//---------------------------------------------------------------------------------------------------------------
//
//  HAUD 2025.12.29
//
//  - fb_LinkedListCtrl
//  -----------------------------
//  - cyclic wrapper composing fb_LinkedList
//  - used to send tickets over the mapping interfaces
//  . Ctrl / State for you to use
//---------------------------------------------------------------------------------------------------------------
FUNCTION_BLOCK fb_Process_LinkedListCtrl
VAR
  _eCheck             : E_LIST_CHECK;
  _eInit              : E_PROGRESS;

  _eCmd,
  _eCmdOld            : E_LIST_CTRL;
  _eState             : E_LIST_STATE;
  _eResult            : e_progress;

  _ItfList            : I_Process_LinkedList;

  _stCtrl             : REFERENCE TO ST_LIST_CTRL;
  _stState            : REFERENCE TO ST_LIST_STATE;

  _stNodeDataInput    : REFERENCE TO ST_LIST_NODE_DATA;   // datafield for you to write(add) your data
  _stNodeDataOutput   : REFERENCE TO ST_LIST_NODE_DATA;   // datafield for you to read (get) your data

  _stNodeDataProcess  : ST_LIST_NODE_DATA;                // local copy of ProcessData

  _stMsg              : ST_Message;
  _eDevice            : e_Device    := e_device.ProcessListCtrl;     // message device identifier
  _MessageLevel       : E_MessageType;

END_VAR

IF NOT Check() 
THEN
  _eInit                          := E_PROGRESS.PROGRESS_INVALID;
  RETURN; 
END_IF


_eCmd                           := _stCtrl.Cmd;
// check for command change
// get state for cmd
IF (_eCmd <> _eCmdOld)
THEN
  _eState                       := Cmd(_eCmd);
  _eCmdOld                      := _eCmd;

  IF (_MessageLevel > E_MessageType.eMessageError)
  THEN
    _stMsg.eType                := E_MessageType.eMessageInfo;
    _stMsg.eSubdevice           := e_Subdevice.Process_LinkedList_Com;
    _stMsg.iErrorNumber         := 0;
    _stMsg.sText                := concat(TO_STRING(_eCmd), ': ');
    _stMsg.sText                := concat(_stMsg.sText,  TO_STRING(_eState));
    f_MessageSet(_stMsg);
  END_IF
END_IF

CASE _eResult
OF
  E_PROGRESS.PROGRESS_INVALID:
    _stState.State              := TO_UINT(_eResult);

  E_PROGRESS.PROGRESS_ERROR:
    _stState.State              := _eState + E_PROGRESS.PROGRESS_ERROR;

  E_PROGRESS.PROGRESS_DONE:
    _stState.State              := _eState + E_PROGRESS.PROGRESS_DONE;

ELSE
  _stState.State                := _eState + _eResult;

  CASE _eState
  OF
    E_LIST_STATE.LIST_STATE_NULL:
      _eResult                  := E_PROGRESS.PROGRESS_DONE;

    E_LIST_STATE.LIST_STATE_INIT:
      _eResult := _eInit        := ListInit (TRUE);

    E_LIST_STATE.LIST_STATE_GET_HEAD:
      _eResult                  := ListGetHead(TRUE);

    E_LIST_STATE.LIST_STATE_GET_TAIL:
      _eResult                  := ListGetTail(TRUE);

    E_LIST_STATE.LIST_STATE_ADD_HEAD:
      _eResult                  := ListAddHead(TRUE);

    E_LIST_STATE.LIST_STATE_ADD_TAIL:
      _eResult                  := ListAddTail(TRUE);

    E_LIST_STATE.LIST_STATE_DEL_HEAD:
      _eResult                  := ListDelHead(TRUE);

    E_LIST_STATE.LIST_STATE_DEL_TAIL:
      _eResult                  := ListDelTail(TRUE);

  ELSE
    _eResult                    := E_PROGRESS.PROGRESS_INVALID;
  END_CASE
END_CASE

_stState.Count                  := _ItfList.Count;
_stState.Free                   := _ItfList.Free;
_stState.Init                   := _eInit;

METHOD Check : bool

IF NOT __ISVALIDREF(_stCtrl)
THEN
  _eCheck                     := E_LIST_CHECK.REFERENCE_CTRL_INVALID;
  RETURN;
END_IF

IF NOT __ISVALIDREF(_stState)
THEN
  _eCheck                     := E_LIST_CHECK.REFERENCE_STATE_INVALID;
  RETURN;
END_IF

IF NOT __ISVALIDREF(_stNodeDataInput)
THEN
  _eCheck                     := E_LIST_CHECK.REFERENCE_DATA_INPUT_INVALID;
  RETURN;
END_IF

IF NOT __ISVALIDREF(_stNodeDataOutput)
THEN
  _eCheck                     := E_LIST_CHECK.REFERENCE_DATA_OUTPUT_INVALID;
  RETURN;
END_IF


_eCheck                       := E_LIST_CHECK.CHECK_DONE;
Check                         := TRUE;
END_METHOD

METHOD Cmd    : E_LIST_STATE;
VAR_INPUT
  Command     : E_LIST_CTRL;
END_VAR
VAR_INST
  _eRslt      : e_progress;
  _eSt        : E_LIST_STATE;
END_VAR
IF NOT Check() THEN RETURN; END_IF

CASE Command
OF
  E_LIST_CTRL.LIST_CTRL_NULL:  // clear all method calls
    _eSt                      := E_LIST_STATE.LIST_STATE_NULL;
    _eResult                  := E_PROGRESS.PROGRESS_INIT;
    _eRslt                    := ListInit    (FALSE);
    _eRslt                    := ListAddHead (FALSE);
    _eRslt                    := ListAddTail (FALSE);
    _eRslt                    := ListDelHead (FALSE);
    _eRslt                    := ListDelTail (FALSE);
    _eRslt                    := ListGetHead (FALSE);
    _eRslt                    := ListGetTail (FALSE);

  E_LIST_CTRL.LIST_CTRL_INIT:  // clear method for initialization
    _eSt                      := E_LIST_STATE.LIST_STATE_INIT;
    _eResult := _eInit        := ListInit (FALSE);

ELSE
  IF NOT (_eInit = E_PROGRESS.PROGRESS_DONE)
  THEN
    // no init, no further commands possible
    _eSt                      := E_LIST_STATE.LIST_STATE_INVALID;

    _stMsg.eType              := E_MessageType.eMessageWarning;
    _stMsg.eSubdevice         := e_Subdevice.Process_LinkedList_Com_Cmd;
    _stMsg.iErrorNumber       := Command;
    _stMsg.sText              := concat('_eInit: ', TO_STRING(_eInit));
    _stMsg.sText              := concat(_stMsg.sText, ': ');
    _stMsg.sText              := concat(_stMsg.sText, TO_STRING(_eSt));
    f_MessageSet(_stMsg);

  ELSE
    CASE Command
    OF
      E_LIST_CTRL.LIST_CTRL_GET_HEAD:
        _eSt                  := E_LIST_STATE.LIST_STATE_GET_HEAD;
        _eResult              := ListGetHead(FALSE);

      E_LIST_CTRL.LIST_CTRL_GET_TAIL:
        _eSt                  := E_LIST_STATE.LIST_STATE_GET_TAIL;
        _eResult              := ListGetTail(FALSE);

      E_LIST_CTRL.LIST_CTRL_ADD_HEAD:
        _eSt                  := E_LIST_STATE.LIST_STATE_ADD_HEAD;
        _stNodeDataProcess      := _stNodeDataInput;
        _eResult              := ListAddHead(FALSE);

      E_LIST_CTRL.LIST_CTRL_ADD_TAIL:
        _eSt                  := E_LIST_STATE.LIST_STATE_ADD_TAIL;
        _stNodeDataProcess      := _stNodeDataInput;
        _eResult              := ListAddTail(FALSE);

      E_LIST_CTRL.LIST_CTRL_DEL_HEAD:
        _eSt                  := E_LIST_STATE.LIST_STATE_DEL_HEAD;
        _eResult              := ListDelHead(FALSE);

      E_LIST_CTRL.LIST_CTRL_DEL_TAIL:
        _eSt                  := E_LIST_STATE.LIST_STATE_DEL_TAIL;
        _eResult              := ListDelTail(FALSE);

    ELSE
        _eSt                  := E_LIST_STATE.LIST_STATE_INVALID;

        _stMsg.eType          := E_MessageType.eMessageError;
        _stMsg.eSubdevice     := e_Subdevice.Process_LinkedList_Com_Cmd;
        _stMsg.iErrorNumber   := Command;
        _stMsg.sText          := concat('Command: ', TO_STRING(Command));
        _stMsg.sText          := concat(_stMsg.sText, ': ');
        _stMsg.sText          := concat(_stMsg.sText, TO_STRING(_eSt));
        f_MessageSet(_stMsg);
    END_CASE
  END_IF
END_CASE

Cmd                           := _eSt;
END_METHOD

PROPERTY Ctrl : REFERENCE TO ST_LIST_CTRL
SET
_stCtrl ref= Ctrl;
END_SET
END_PROPERTY

PROPERTY ItfList : I_Process_LinkedList
SET
_ItfList := ItfList;
END_SET
END_PROPERTY

METHOD ListAddHead  : e_progress
VAR_INPUT
  Execute           : BOOL;
END_VAR
VAR_INST
  _ListResult       : ST_PROCESS_LIST_RESULT;
  _nErrorId         : UDINT;
  _eState           : E_PROGRESS;
END_VAR
//-----------------------------------------------------------------------------
IF NOT Execute 
THEN 
	_eState                       := E_PROGRESS.PROGRESS_INIT; 
END_IF 
//-----------------------------------------------------------------------------
IF NOT Check() 
THEN 
	ListAddHead                   := E_PROGRESS.PROGRESS_ERROR; 
	RETURN; 
END_IF
//-----------------------------------------------------------------------------
//-----------------------------------------------------------------------------
CASE _eState
OF
  E_PROGRESS.PROGRESS_INIT:
    IF Execute
    THEN
      _nErrorId                 := 0;
      _eState                   := E_PROGRESS.PROGRESS_BUSY;
    END_IF
END_CASE
//-----------------------------------------------------------------------------
//-----------------------------------------------------------------------------
CASE _eState
OF
  E_PROGRESS.PROGRESS_BUSY:
    _eState                     := E_PROGRESS.PROGRESS_PREPARE;
    _ListResult                 := _ItfList.AddHeadValue(_stNodeDataProcess.ProcessData);
END_CASE
//-----------------------------------------------------------------------------
//-----------------------------------------------------------------------------
CASE _eState
OF
  E_PROGRESS.PROGRESS_PREPARE:

    IF (_ListResult.wState <> 0)
    THEN
      _eState                   := E_PROGRESS.PROGRESS_ERROR;
      _nErrorId                 := _ListResult.wState;

      _stMsg.eType              := E_MessageType.eMessageError;
      _stMsg.eSubdevice         := e_Subdevice.Process_LinkedList_Com_AddHead;
      _stMsg.iErrorNumber       := _nErrorId;
      _stMsg.sText              := '';
      _stMsg.sText              := concat(_stMsg.sText, TO_STRING(_eState));
      f_MessageSet(_stMsg);

    ELSE
      _eState                   := E_PROGRESS.PROGRESS_DONE;

      IF (_MessageLevel > E_MessageType.eMessageError)
      THEN
        _stMsg.eType            := E_MessageType.eMessageInfo;
        _stMsg.eSubdevice       := e_Subdevice.Process_LinkedList_Com_AddHead;
        _stMsg.iErrorNumber     := 0;
        _stMsg.sText            := '';
        _stMsg.sText            := concat(_stMsg.sText, TO_STRING(_eState));
        f_MessageSet(_stMsg);
      END_IF
    END_IF
END_CASE
//-----------------------------------------------------------------------------
//-----------------------------------------------------------------------------

ListAddHead                     := _eState;
END_METHOD

METHOD ListAddTail  : e_progress
VAR_INPUT
  Execute           : BOOL;
END_VAR
VAR_INST
  _ListResult       : ST_PROCESS_LIST_RESULT;
  _nErrorId         : UDINT;
  _eState           : E_PROGRESS;
END_VAR
//-----------------------------------------------------------------------------
IF NOT Execute 
THEN 
	_eState                       := E_PROGRESS.PROGRESS_INIT; 
END_IF 
//-----------------------------------------------------------------------------
IF NOT Check() 
THEN 
	ListAddTail                   := E_PROGRESS.PROGRESS_ERROR; 
	RETURN; 
END_IF
//-----------------------------------------------------------------------------
//-----------------------------------------------------------------------------
CASE _eState
OF
  E_PROGRESS.PROGRESS_INIT:
    IF Execute
    THEN
      _nErrorId                 := 0;
      _eState                   := E_PROGRESS.PROGRESS_BUSY;
    END_IF
END_CASE
//-----------------------------------------------------------------------------
//-----------------------------------------------------------------------------
CASE _eState
OF
  E_PROGRESS.PROGRESS_BUSY:
    _eState                     := E_PROGRESS.PROGRESS_PREPARE;
    _ListResult                 := _ItfList.AddTailValue(_stNodeDataProcess.ProcessData);
END_CASE
//-----------------------------------------------------------------------------
//-----------------------------------------------------------------------------
CASE _eState
OF
  E_PROGRESS.PROGRESS_PREPARE:

    IF (_ListResult.wState <> 0)
    THEN
      _eState                   := E_PROGRESS.PROGRESS_ERROR;
      _nErrorId                 := _ListResult.wState;

      _stMsg.eType              := E_MessageType.eMessageError;
      _stMsg.eSubdevice         := e_Subdevice.Process_LinkedList_Com_AddTail;
      _stMsg.iErrorNumber       := _nErrorId;
      _stMsg.sText              := '';
      _stMsg.sText              := concat(_stMsg.sText, TO_STRING(_eState));
      f_MessageSet(_stMsg);

    ELSE
      _eState                   := E_PROGRESS.PROGRESS_DONE;

      IF (_MessageLevel > E_MessageType.eMessageError)
      THEN
        _stMsg.eType            := E_MessageType.eMessageInfo;
        _stMsg.eSubdevice       := e_Subdevice.Process_LinkedList_Com_AddTail;
        _stMsg.iErrorNumber     := 0;
        _stMsg.sText            := '';
        _stMsg.sText            := concat(_stMsg.sText, TO_STRING(_eState));
        f_MessageSet(_stMsg);
      END_IF
    END_IF
END_CASE
//-----------------------------------------------------------------------------
//-----------------------------------------------------------------------------

ListAddTail                     := _eState;
END_METHOD

METHOD ListDelHead  : e_progress
VAR_INPUT
  Execute           : BOOL;
END_VAR
VAR_INST
  _ListResult       : ST_PROCESS_LIST_RESULT;
  _nErrorId         : UDINT;
  _eState           : E_PROGRESS;
END_VAR
//-----------------------------------------------------------------------------
IF NOT Execute 
THEN 
	_eState                       := E_PROGRESS.PROGRESS_INIT; 
END_IF 
//-----------------------------------------------------------------------------
IF NOT Check() 
THEN 
	ListDelHead                   := E_PROGRESS.PROGRESS_ERROR; 
	RETURN; 
END_IF
//-----------------------------------------------------------------------------
//-----------------------------------------------------------------------------
CASE _eState
OF
  E_PROGRESS.PROGRESS_INIT:
    IF Execute
    THEN
      _nErrorId                 := 0;
      _eState                   := E_PROGRESS.PROGRESS_BUSY;
    END_IF
END_CASE
//-----------------------------------------------------------------------------
//-----------------------------------------------------------------------------
CASE _eState
OF
  E_PROGRESS.PROGRESS_BUSY:
    _eState                     := E_PROGRESS.PROGRESS_PREPARE;
    _ListResult                 := _ItfList.RemoveHeadValue();
END_CASE
//-----------------------------------------------------------------------------
//-----------------------------------------------------------------------------
CASE _eState
OF
  E_PROGRESS.PROGRESS_PREPARE:

    IF (_ListResult.wState <> 0)
    THEN
      _eState                   := E_PROGRESS.PROGRESS_ERROR;
      _nErrorId                 := _ListResult.wState;

      _stMsg.eType              := E_MessageType.eMessageError;
      _stMsg.eSubdevice         := e_Subdevice.Process_LinkedList_Com_DelHead;
      _stMsg.iErrorNumber       := _nErrorId;
      _stMsg.sText              := '';
      _stMsg.sText              := concat(_stMsg.sText, TO_STRING(_eState));
      f_MessageSet(_stMsg);

    ELSE
      _eState                   := E_PROGRESS.PROGRESS_DONE;

      IF (_MessageLevel > E_MessageType.eMessageError)
      THEN
        _stMsg.eType            := E_MessageType.eMessageInfo;
        _stMsg.eSubdevice       := e_Subdevice.Process_LinkedList_Com_DelHead;
        _stMsg.iErrorNumber     := 0;
        _stMsg.sText            := '';
        _stMsg.sText            := concat(_stMsg.sText, TO_STRING(_eState));
        f_MessageSet(_stMsg);
      END_IF
    END_IF
END_CASE
//-----------------------------------------------------------------------------
//-----------------------------------------------------------------------------

ListDelHead                     := _eState;
END_METHOD

METHOD ListDelTail  : e_progress
VAR_INPUT
  Execute           : BOOL;
END_VAR
VAR_INST
  _ListResult       : ST_PROCESS_LIST_RESULT;
  _nErrorId         : UDINT;
  _eState           : E_PROGRESS;
END_VAR
//-----------------------------------------------------------------------------
IF NOT Execute 
THEN 
	_eState                       := E_PROGRESS.PROGRESS_INIT; 
END_IF 
//-----------------------------------------------------------------------------
IF NOT Check() 
THEN 
	ListDelTail                   := E_PROGRESS.PROGRESS_ERROR; 
	RETURN; 
END_IF
//-----------------------------------------------------------------------------
//-----------------------------------------------------------------------------
CASE _eState
OF
  E_PROGRESS.PROGRESS_INIT:
    IF Execute
    THEN
      _nErrorId                 := 0;
      _eState                   := E_PROGRESS.PROGRESS_BUSY;
    END_IF
END_CASE
//-----------------------------------------------------------------------------
//-----------------------------------------------------------------------------
CASE _eState
OF
  E_PROGRESS.PROGRESS_BUSY:
    _eState                     := E_PROGRESS.PROGRESS_PREPARE;
    _ListResult                 := _ItfList.RemoveTailValue();
END_CASE
//-----------------------------------------------------------------------------
//-----------------------------------------------------------------------------
CASE _eState
OF
  E_PROGRESS.PROGRESS_PREPARE:

    IF (_ListResult.wState <> 0)
    THEN
      _eState                   := E_PROGRESS.PROGRESS_ERROR;
      _nErrorId                 := _ListResult.wState;

      _stMsg.eType              := E_MessageType.eMessageError;
      _stMsg.eSubdevice         := e_Subdevice.Process_LinkedList_Com_DelTail;
      _stMsg.iErrorNumber       := _nErrorId;
      _stMsg.sText              := '';
      _stMsg.sText              := concat(_stMsg.sText, TO_STRING(_eState));
      f_MessageSet(_stMsg);

    ELSE
      _eState                   := E_PROGRESS.PROGRESS_DONE;

      IF (_MessageLevel > E_MessageType.eMessageError)
      THEN
        _stMsg.eType            := E_MessageType.eMessageInfo;
        _stMsg.eSubdevice       := e_Subdevice.Process_LinkedList_Com_DelTail;
        _stMsg.iErrorNumber     := 0;
        _stMsg.sText            := '';
        _stMsg.sText            := concat(_stMsg.sText, TO_STRING(_eState));
        f_MessageSet(_stMsg);
      END_IF
    END_IF
END_CASE
//-----------------------------------------------------------------------------
//-----------------------------------------------------------------------------

ListDelTail                     := _eState;
END_METHOD

METHOD ListGetHead  : e_progress
VAR_INPUT
  Execute           : BOOL;
END_VAR
VAR_INST
  _ListResult       : ST_PROCESS_LIST_RESULT;
  _nErrorId         : UDINT;
  _eState           : E_PROGRESS;
END_VAR
//-----------------------------------------------------------------------------
IF NOT Execute 
THEN 
	_eState                         := E_PROGRESS.PROGRESS_INIT; 
END_IF 
//-----------------------------------------------------------------------------
IF NOT Check() 
THEN 
	ListGetHead                     := E_PROGRESS.PROGRESS_ERROR; 
	RETURN; 
END_IF
//-----------------------------------------------------------------------------
//-----------------------------------------------------------------------------
CASE _eState
OF
  E_PROGRESS.PROGRESS_INIT:
    IF Execute
    THEN
      _nErrorId                   := 0;
      _eState                     := E_PROGRESS.PROGRESS_BUSY;
    END_IF
END_CASE
//-----------------------------------------------------------------------------
//-----------------------------------------------------------------------------
CASE _eState
OF
  E_PROGRESS.PROGRESS_BUSY:
    _eState                       := E_PROGRESS.PROGRESS_PREPARE;
    _ListResult                   := _ItfList.GetHead();
END_CASE
//-----------------------------------------------------------------------------
//-----------------------------------------------------------------------------
CASE _eState
OF
  E_PROGRESS.PROGRESS_PREPARE:

    IF (_ListResult.wState <> 0)
    THEN
      _eState                     := E_PROGRESS.PROGRESS_ERROR;
      _nErrorId                   := _ListResult.wState;

      _stMsg.eType                := E_MessageType.eMessageError;
      _stMsg.eSubdevice           := e_Subdevice.Process_LinkedList_Com_GetHead;
      _stMsg.iErrorNumber         := _nErrorId;
      _stMsg.sText                := '';
      _stMsg.sText                := concat(_stMsg.sText, TO_STRING(_eState));
      f_MessageSet(_stMsg);

    ELSE
      _stNodeDataProcess.ProcessData:= _ListResult.stData;
      _stNodeDataOutput             := _stNodeDataProcess;

      _eState                     := E_PROGRESS.PROGRESS_DONE;

      IF (_MessageLevel > E_MessageType.eMessageError)
      THEN
        _stMsg.eType              := E_MessageType.eMessageInfo;
        _stMsg.eSubdevice         := e_Subdevice.Process_LinkedList_Com_GetHead;
        _stMsg.iErrorNumber       := 0;
        _stMsg.sText              := '';
        _stMsg.sText              := concat(_stMsg.sText, TO_STRING(_eState));
        f_MessageSet(_stMsg);
      END_IF
    END_IF
END_CASE
//-----------------------------------------------------------------------------
//-----------------------------------------------------------------------------

ListGetHead                       := _eState;
END_METHOD

METHOD ListGetTail  : e_progress
VAR_INPUT
  Execute           : BOOL;
END_VAR
VAR_INST
  _ListResult       : ST_PROCESS_LIST_RESULT;
  _nErrorId         : UDINT;
  _eState           : E_PROGRESS;
END_VAR
//-----------------------------------------------------------------------------
IF NOT Execute 
THEN 
	_eState                         := E_PROGRESS.PROGRESS_INIT; 
END_IF 
//-----------------------------------------------------------------------------
IF NOT Check() 
THEN 
	ListGetTail                     := E_PROGRESS.PROGRESS_ERROR; 
	RETURN; 
END_IF
//-----------------------------------------------------------------------------
//-----------------------------------------------------------------------------
CASE _eState
OF
  E_PROGRESS.PROGRESS_INIT:
    IF Execute
    THEN
      _nErrorId                   := 0;
      _eState                     := E_PROGRESS.PROGRESS_BUSY;
    END_IF
END_CASE
//-----------------------------------------------------------------------------
//-----------------------------------------------------------------------------
CASE _eState
OF
  E_PROGRESS.PROGRESS_BUSY:
    _eState                       := E_PROGRESS.PROGRESS_PREPARE;
    _ListResult                   := _ItfList.GetTail();
END_CASE
//-----------------------------------------------------------------------------
//-----------------------------------------------------------------------------
CASE _eState
OF
  E_PROGRESS.PROGRESS_PREPARE:

    IF (_ListResult.wState <> 0)
    THEN
      _eState                     := E_PROGRESS.PROGRESS_ERROR;
      _nErrorId                   := _ListResult.wState;

      _stMsg.eType                := E_MessageType.eMessageError;
      _stMsg.eSubdevice           := e_Subdevice.Process_LinkedList_Com_GetTail;
      _stMsg.iErrorNumber         := _nErrorId;
      _stMsg.sText                := '';
      _stMsg.sText                := concat(_stMsg.sText, TO_STRING(_eState));
      f_MessageSet(_stMsg);

    ELSE
      _stNodeDataProcess.ProcessData:= _ListResult.stData;
      _stNodeDataOutput             := _stNodeDataProcess;

      _eState                     := E_PROGRESS.PROGRESS_DONE;

      IF (_MessageLevel > E_MessageType.eMessageError)
      THEN
        _stMsg.eType              := E_MessageType.eMessageInfo;
        _stMsg.eSubdevice         := e_Subdevice.Process_LinkedList_Com_GetTail;
        _stMsg.iErrorNumber       := 0;
        _stMsg.sText              := '';
        _stMsg.sText              := concat(_stMsg.sText, TO_STRING(_eState));
        f_MessageSet(_stMsg);
      END_IF
    END_IF
END_CASE
//-----------------------------------------------------------------------------
//-----------------------------------------------------------------------------

ListGetTail                       := _eState;
END_METHOD

METHOD ListInit  : e_progress
VAR_INPUT
  Execute           : BOOL;
END_VAR
VAR_INST
  _ListResult       : BOOL;

  _nErrorId         : UDINT;
  _eState           : E_PROGRESS;
END_VAR
//-----------------------------------------------------------------------------
IF NOT Execute 
THEN 
	_eState                       := E_PROGRESS.PROGRESS_INIT; 
END_IF 
//-----------------------------------------------------------------------------
IF NOT Check() 
THEN 
	ListInit                      := E_PROGRESS.PROGRESS_ERROR; 
	RETURN; 
END_IF
//-----------------------------------------------------------------------------
//-----------------------------------------------------------------------------
CASE _eState
OF
  E_PROGRESS.PROGRESS_INIT:
    IF Execute
    THEN
      _nErrorId                 := 0;
      _eState                   := E_PROGRESS.PROGRESS_BUSY;
    END_IF
END_CASE
//-----------------------------------------------------------------------------
//-----------------------------------------------------------------------------
CASE _eState
OF
  E_PROGRESS.PROGRESS_BUSY:
    _eState                     := E_PROGRESS.PROGRESS_PREPARE;
    _ListResult                 := _ItfList.InitList();
END_CASE
//-----------------------------------------------------------------------------
//-----------------------------------------------------------------------------
CASE _eState
OF
  E_PROGRESS.PROGRESS_PREPARE:

    IF NOT (_ListResult)
    THEN
      _eState                   := E_PROGRESS.PROGRESS_ERROR;
      _nErrorId                 := 666;

      _stMsg.eType              := E_MessageType.eMessageError;
      _stMsg.eSubdevice         := e_Subdevice.Process_LinkedList_Com_Init;
      _stMsg.iErrorNumber       := _nErrorId;
      _stMsg.sText              := '';
      _stMsg.sText              := concat(_stMsg.sText, TO_STRING(_eState));
      f_MessageSet(_stMsg);

    ELSE
      _eState                   := E_PROGRESS.PROGRESS_DONE;

      IF (_MessageLevel > E_MessageType.eMessageError)
      THEN
        _stMsg.eType            := E_MessageType.eMessageInfo;
        _stMsg.eSubdevice       := e_Subdevice.Process_LinkedList_Com_Init;
        _stMsg.iErrorNumber     := 0;
        _stMsg.sText            := '';
        _stMsg.sText            := concat(_stMsg.sText, TO_STRING(_eState));
        f_MessageSet(_stMsg);
      END_IF
    END_IF
END_CASE
//-----------------------------------------------------------------------------
//-----------------------------------------------------------------------------

ListInit                        := _eState;
END_METHOD

PROPERTY MessageLevel : e_MessageType
GET
MessageLevel := _MessageLevel;
END_GET
SET
_MessageLevel := MessageLevel;
END_SET
END_PROPERTY

PROPERTY NodeDataInput : reference to st_list_node_data
SET
_stNodeDataInput REF= NodeDataInput;
END_SET
END_PROPERTY

PROPERTY NodeDataOutput : reference to st_list_node_data
SET
_stNodeDataOutput REF= NodeDataOutput;
END_SET
END_PROPERTY

PROPERTY State : REFERENCE TO ST_LIST_STATE
SET
_stState ref= State;
END_SET
END_PROPERTY

END_FUNCTION_BLOCK

(* stored: Version 1.1.0.1, ProductVersion 3.1.4026.13
   POU fb_Process_LinkedListCtrl: Id {1e362c19-c72b-4969-8606-a64fee7d78f2}, SpecialFunc None
   Folder properties: Id {518ca38e-66ef-47e5-8606-899395a9d769}
   Method Check: Id {0371c119-9a73-460c-8212-6d13e14ec1d9}
   Method Cmd: Id {4f69743f-0e81-471d-a6c4-04e7add4ce79}
   Property Ctrl: Id {f4f51022-2c81-4010-9182-895442660b74}
   Set Set: Id {1b5bb6bb-97b3-425a-ade6-eca4c904a88f}
   Property ItfList: Id {91f5f846-19df-4ced-948e-76e51e5a6ab0}
   Set Set: Id {9d9b2349-2db3-4c28-8c9c-3f23151489bf}
   Method ListAddHead: Id {f34a8244-a618-4bfb-9cab-04407908eb4b}
   Method ListAddTail: Id {4fd88cb8-55e3-4bd5-80b6-93cbd0833dc5}
   Method ListDelHead: Id {feb5114c-bee1-43c2-a13a-d20c6335ad66}
   Method ListDelTail: Id {076a7056-19b2-438a-831f-271e9b24e63a}
   Method ListGetHead: Id {97e43b81-2c21-4b83-bcfb-3dd1f7b66923}
   Method ListGetTail: Id {c02e2ffb-8c63-4d93-97f1-137e2b86b1e9}
   Method ListInit: Id {64a98cca-bc34-4981-a01e-0aab4fe173f8}
   Property MessageLevel: Id {033a2630-8113-40c4-80f0-db1e15997cce}
   Get Get: Id {bca12089-434b-4ce3-a7ad-bd084c8f521d}
   Set Set: Id {d4dbae17-efea-44c4-b980-4aba6c0ceca5}
   Property NodeDataInput: Id {a932ac25-db29-4c32-8bb7-ff9aacd7ff06}
   Set Set: Id {96376859-7792-4c3b-8060-638a44bf9898}
   Property NodeDataOutput: Id {7b01a671-a20a-46af-80fd-e38aeb9415f1}
   Set Set: Id {462758c7-4e52-425d-a7ad-c663e6fdd4b2}
   Property State: Id {3782915e-99c4-4f77-b8a0-88fc53d343b5}
   Set Set: Id {834b3722-d7fe-4b96-ab4c-7705b3b2c74f} *)
